INTERFACE I_CH_LIST

//DEBUG only. View content for easy debug. Do not use this property
{attribute 'monitoring':='call'}
PROPERTY Content : REFERENCE TO ARRAY [1..BaseParameterlist.MAX_OBJECTS] OF I_CH_Object
GET
END_GET
END_PROPERTY

METHOD PUBLIC FindLUID : I_CH_OBJECT
VAR_INPUT
	sLUID	: STRING;
END_VAR
END_METHOD

METHOD FindOID : I_CH_OBJECT
VAR_INPUT
	nOID	: OTCID;
END_VAR
END_METHOD

METHOD FindOIDString : I_CH_OBJECT
VAR_INPUT
	sOID	: STRING;
END_VAR
END_METHOD

METHOD PUBLIC GetNextObject : I_CH_Object
VAR_INPUT
END_VAR
END_METHOD

METHOD GetObjectWithHighestNumber : I_CH_Object
END_METHOD

METHOD GetObjectWithLowestNumber : I_CH_Object
END_METHOD

METHOD GetRandomObject : I_CH_Object
VAR_INPUT
END_VAR
END_METHOD

METHOD PUBLIC HasNextObject : BOOL
VAR_INPUT
END_VAR
END_METHOD

{attribute 'monitoring':='call'}
PROPERTY PUBLIC IsEmpty : BOOL
GET
END_GET
END_PROPERTY

{attribute 'monitoring':='call'}
PROPERTY PUBLIC IsFull : BOOL
GET
END_GET
END_PROPERTY

METHOD PUBLIC LUIDInList : BOOL
VAR_INPUT
	sLUID	: STRING;
END_VAR
END_METHOD

METHOD PUBLIC ObjectInList : BOOL
VAR_INPUT
	iChObject	: I_CH_Object;
END_VAR
END_METHOD

METHOD PUBLIC OIDInList : BOOL
VAR_INPUT
	nOID	: OTCID;
END_VAR
END_METHOD

METHOD RemoveAllDuplicateObjects : HRESULT
VAR_INPUT
END_VAR
END_METHOD

METHOD PUBLIC ResetIterator : BOOL
VAR_INPUT
END_VAR
END_METHOD

//Restore the iterator to the value before the last reset. This is necessary if several while loops are placed inside each other
METHOD PUBLIC RestoreIterator : BOOL
VAR_INPUT
END_VAR
END_METHOD

{attribute 'monitoring':='call'}
PROPERTY PUBLIC Size : UDINT
GET
END_GET
END_PROPERTY

END_INTERFACE

(* stored: Version 1.1.0.1, ProductVersion 3.1.4024.12
   Itf I_CH_LIST: Id {d81cb508-fdd5-4139-a740-4def79be0c9c}
   Folder Debug: Id {3f0a098f-0460-439d-a8f7-37aa7612e213}
   Folder ID: Id {b5bee6b3-f34b-4142-822a-3bcf3bc4785b}
   Folder Iterator: Id {7a7c31ed-bfb1-4340-bc39-4f11a11e3794}
   Folder List: Id {ab4ecb65-114f-4800-8f52-0f0cb42c1aa5}
   Folder Object: Id {f7f4e7ee-8120-414e-9a76-54cfdf0852c8}
   Folder Sort: Id {35d21c57-0fe2-48d2-a4bf-54135e98546d}
   Property Content: Id {fb93fbe7-0b6a-45f9-ade1-a986d6c8fe07}
   Get Get: Id {9a56c5e0-863f-4eb7-a4ee-e4283ff43e87}
   Method FindLUID: Id {b1c63aa2-f24f-4f14-9da7-0d917025b72e}
   Method FindOID: Id {0f77295a-574e-4005-8b7a-219431a3336f}
   Method FindOIDString: Id {56977772-656e-4bac-acda-b7157561a0a9}
   Method GetNextObject: Id {1c7b796b-f015-453e-ad77-33118df7f431}
   Method GetObjectWithHighestNumber: Id {512eb182-fcc3-4841-980b-312825679c4e}
   Method GetObjectWithLowestNumber: Id {fe0aba4e-8ef2-438c-a526-44a29387eb4a}
   Method GetRandomObject: Id {c3d5e421-67b1-44a7-8dc5-765066f5a1a3}
   Method HasNextObject: Id {594b4e43-9d17-49e3-8008-0d53d7e8f475}
   Property IsEmpty: Id {d3abda63-2a30-4497-96f0-7df6765ad498}
   Get Get: Id {79cb8286-ac05-4e44-a30e-a9d78018dbd0}
   Property IsFull: Id {6c230d12-db05-4952-a351-45df63272d31}
   Get Get: Id {70af465e-62e3-43fc-9513-246efd9b9f1a}
   Method LUIDInList: Id {991f0cc3-7ee6-4a66-9716-0f0e5d809c37}
   Method ObjectInList: Id {e1aa04d1-835b-4b84-8b94-235211f2913d}
   Method OIDInList: Id {a5f3bce5-474f-4e1c-a60e-a22084904f90}
   Method RemoveAllDuplicateObjects: Id {43a6597e-7b09-42a5-b512-ddcf6b7559c7}
   Method ResetIterator: Id {bab1e98b-f88f-4090-a6c9-84a76c2767bd}
   Method RestoreIterator: Id {33f0a221-2302-4c17-ac96-3f011c5c97be}
   Property Size: Id {b6426dfa-8408-4c4c-946b-84af6c72a15a}
   Get Get: Id {1b00da5e-dad4-4d63-8d1e-dacc49874e60} *)
